FUNCTION_BLOCK FB_HomeNC IMPLEMENTS I_Home
VAR
    {attribute 'no_copy'}
    AxisRef : REFERENCE TO AXIS_REF;
    iMotionLogger : I_MotionLogger;
    iLimSwStatus : I_LimSwStatus;
    fbMcHome : MC_Home;
    eHomeState : (WaitingHome, Homing);


    fOffset  : LREAL;
    fPosition	: LREAL;
    bFirstDirection: BOOL;
    rtDone				: R_TRIG;
    rtAborted : R_TRIG;
    sMessage : T_MAXSTRING;
    fbMcSetPos: MC_SetPosition;
    fbMcJog: MC_Jog;
    rtExec: R_TRIG;
    ftExec: F_TRIG;
    bCommandMoveHome : BOOL;
    bAtHome: BOOL;
    bMove: BOOL;
    eHomeMode: E_EpicsHomeCmd :=E_EpicsHomeCmd.NONE;

END_VAR

IF NOT __ISVALIDREF(AxisRef) THEN
    RETURN;
END_IF

CASE eHomeMode OF
    E_EpicsHomeCmd.LOW_LIMIT:
        fbMcHome.HomingMode := MC_HomingMode.MC_DefaultHoming;
        fbMcHome.Options.SearchDirection := MC_Direction.MC_Negative_Direction;
        fbMcHome.Options.SyncDirection := MC_Direction.MC_Positive_Direction;
        fbMcHome.Options.ClearPositionLag := TRUE;
        fbMcHome.bCalibrationCam := NOT iLimSwStatus.LimBackward;
        bMove := TRUE;
    E_EpicsHomeCmd.HIGH_LIMIT:
        fbMcHome.HomingMode := MC_HomingMode.MC_DefaultHoming;
        fbMcHome.Options.SearchDirection := MC_Direction.MC_Positive_Direction;
        fbMcHome.Options.SyncDirection := MC_Direction.MC_Negative_Direction;
        fbMcHome.Options.ClearPositionLag := TRUE;
        fbMcHome.bCalibrationCam := NOT iLimSwStatus.LimForward;
    E_EpicsHomeCmd.HOME_VIA_LOW:
        fbMcHome.HomingMode := MC_HomingMode.MC_DefaultHoming;
        fbMcHome.Options.SearchDirection := MC_Direction.MC_Negative_Direction;
        fbMcHome.Options.SyncDirection := MC_Direction.MC_Positive_Direction;
        fbMcHome.Options.ClearPositionLag := TRUE;
        fbMcHome.bCalibrationCam := iLimSwStatus.LimHome;
    E_EpicsHomeCmd.HOME_VIA_HIGH:
        fbMcHome.HomingMode := MC_HomingMode.MC_DefaultHoming;
        fbMcHome.Options.SearchDirection := MC_Direction.MC_Positive_Direction;
        fbMcHome.Options.SyncDirection := MC_Direction.MC_Negative_Direction;
        fbMcHome.Options.ClearPositionLag := TRUE;
        fbMcHome.bCalibrationCam := iLimSwStatus.LimHome;
    E_EpicsHomeCmd.ABSOLUTE_SET:
        fbMcHome.HomingMode := MC_HomingMode.MC_Direct;
        fbMcHome.Options.SearchDirection := MC_Direction.MC_Undefined_Direction;
        fbMcHome.Options.SyncDirection := MC_Direction.MC_Undefined_Direction;
        fbMcHome.Options.ClearPositionLag := TRUE;
END_CASE

fbMcHome(Axis := AxisRef);

PROPERTY Aborted : BOOL
GET
Aborted := fbMcHome.CommandAborted;
END_GET
END_PROPERTY

PROPERTY Active : BOOL
GET
Active := fbMcHome.Active;
END_GET
END_PROPERTY

PROPERTY Busy : BOOL
GET
Busy := fbMcHome.Busy;
END_GET
END_PROPERTY

METHOD PUBLIC CallAfterInit
VAR_INPUT
    AxisRef : REFERENCE TO AXIS_REF;
    iMotionLogger : I_MotionLogger;
    iLimSwStatus : I_LimSwStatus;
END_VAR
THIS^.AxisRef REF= AxisRef;
THIS^.iMotionLogger := iMotionLogger;
THIS^.iLimSwStatus:= iLimSwStatus;
END_METHOD

PROPERTY Done : BOOL
GET
IF THIS^.eHomeMode <> E_EpicsHomeCmd.NONE THEN
    Done :=fbMcHome.Done;
ELSE
    Done :=TRUE;
END_IF
END_GET
END_PROPERTY

PROPERTY Error : BOOL
GET
Error := fbMcHome.Error;
END_GET
END_PROPERTY

PROPERTY ErrorID : UDINT
GET
ErrorID := fbMcHome.ErrorID;
END_GET
END_PROPERTY

//FB_Init is always available implicitly and it is used primarily for initialization.
//The return value is not evaluated. For a specific influence, you can also declare the
//methods explicitly and provide additional code there with the standard initialization
//code. You can evaluate the return value.
METHOD FB_Init: BOOL
VAR_INPUT
    bInitRetains: BOOL; // TRUE: the retain variables are initialized (reset warm / reset cold)
    bInCopyCode: BOOL;  // TRUE: the instance will be copied to the copy code afterward (online change)
    AxisRef : REFERENCE TO AXIS_REF;
    iMotionLogger : I_MotionLogger;
    iLimSwStatus : I_LimSwStatus;
END_VAR
THIS^.AxisRef REF= AxisRef;
THIS^.iMotionLogger := iMotionLogger;
THIS^.iLimSwStatus:= iLimSwStatus;
END_METHOD

METHOD  Home
VAR_INPUT
    Position        : LREAL         := DEFAULT_HOME_POSITION;
    BufferMode      : MC_BufferMode;
END_VAR
IF THIS^.eHomeMode = E_EpicsHomeCmd.NONE THEN
    RETURN;
END_IF

fbMcHome(Execute := FALSE, Axis := THIS^.AxisRef);



fbMcHome(	Execute := TRUE,
            Axis := THIS^.AxisRef,
            Position:=Position,
            BufferMode:=BufferMode);

eHomeState := Homing;
END_METHOD

PROPERTY Message : T_MAXSTRING
GET
Message := sMessage;
END_GET
END_PROPERTY

PROPERTY Mode : E_EpicsHomeCmd
GET
Mode := eHomeMode;
END_GET
SET
eHomeMode := Mode;
END_SET
END_PROPERTY

PROPERTY Offset : LREAL
SET
fOffset := Offset;
END_SET
END_PROPERTY

PROPERTY Position : LREAL
SET
fPosition := Position;
END_SET
END_PROPERTY

END_FUNCTION_BLOCK

(* stored: Version 1.1.0.1
   POU FB_HomeNC: Id {970a142c-358e-492f-9cec-3782954ac4db}, SpecialFunc None
   Property Aborted: Id {b3440598-2192-4aa3-bd94-648810782f1d}
   Get Get: Id {6a45fc91-d1f8-4045-827a-687d21932173}
   Property Active: Id {4386ac45-3e88-4c79-8d18-81c7e83c1e8e}
   Get Get: Id {bdd5f606-f201-4f1a-9491-5ed9fc2ed98d}
   Property Busy: Id {c7e43be2-48b0-438b-8ceb-465d60425bfc}
   Get Get: Id {cb0740bd-cd32-462e-8d30-3401b18588d5}
   Method CallAfterInit: Id {bf0efffc-cb26-4144-93d7-4a53b23636d4}
   Property Done: Id {a400b97e-6245-4667-8036-7fb53f8ce97f}
   Get Get: Id {aef52b53-9bff-4703-970f-52b560ffba73}
   Property Error: Id {d9029227-7d8c-4426-821a-d46327fbfa6d}
   Get Get: Id {4884c9e1-0ab0-469e-aae8-b83b96b6f583}
   Property ErrorID: Id {cf64e9b6-c8bf-4aa1-9fa1-b62063c78b03}
   Get Get: Id {e14def51-9c37-4182-ba09-611583cf679e}
   Method FB_Init: Id {36203808-aa8e-419d-b89f-47cad560b581}
   Method Home: Id {bc450e32-fe3c-4fef-961a-7ec21133b561}
   Property Message: Id {50dd0817-9d23-4b27-bd5b-fe17ea82eb6e}
   Get Get: Id {5582f213-525c-49f8-9472-dcc0e7068f61}
   Property Mode: Id {bacfc68b-674d-49fb-a838-6a7b08d66c8b}
   Get Get: Id {018ebc11-483b-4d91-b1ca-54274e9fa554}
   Set Set: Id {d7a9685a-e050-4fa2-92a8-d25079a18728}
   Property Offset: Id {48496da5-ced9-4c7a-88b4-656a32aa685b}
   Set Set: Id {0ef7a418-62f9-4e76-9f2c-837b987f3900}
   Property Position: Id {afef80c7-a1a3-4197-a7a0-d9553542477a}
   Set Set: Id {6ac419d4-6add-4703-8089-625e0296877b} *)
